GLOBALCONSTANTS HANDLE (* Global constants *)
  (* Standard: 61499-1 *)
  (* Version 1.0, 2025-09-04, Franz Höpfinger *)
  PACKAGE isobus::pgn;
  IMPORT eclipse4diac::core::TypeHash;
  VAR_GLOBAL CONSTANT
    UNVALID : INT := (-1);
    GLOBAL : INT := 32767; (* < \brief 0xFFFF Invalid or unused handle *)
  END_VAR
END_GLOBALCONSTANTS
